// TIA Portal V20 export
DATA_BLOCK "GLOBAL_IDENT_DATA_DB"   // DB207
{ S7_Optimized_Access := 'TRUE' }
AUTHOR : Tesla
FAMILY : Ident
VERSION : 1.0
// stored: AutoNumber false, MemoryReserve 100
   VAR
      Reader { ExternalAccessible := 'False'; ExternalVisible := 'False'; ExternalWritable := 'False'; S7_SetPoint := 'True'} : Array[0.."No_Reader"] of "IDENT_RW_BYTE_DAT_UDT";
   END_VAR
BEGIN
END_DATA_BLOCK
